% RSLogix 500 project DDE_Conecction_Excel.RSS, saved by version 8.30.00.16 %
PROJECT "UNTITLED"    % processor: Bul.1763 MicroLogix 1100 Series B %

PROGRAM FILES
  LAD 2 "MAIN"  4 rungs
  LAD 3 "DDE EXCEL"  31 rungs

DATA FILES
  O0 OUTPUT  4 elements
  I1 INPUT  6 elements
  S2 STATUS  66 elements
  B3 BINARY  2 elements
  T4 TIMER  8 elements
  C5 COUNTER  4 elements
  R6 CONTROL  1 elements
  N7 INTEGER  9 elements
  F8 FLOAT  1 elements
  ST9 STRINGS  9 elements

LADDER 2 "MAIN"
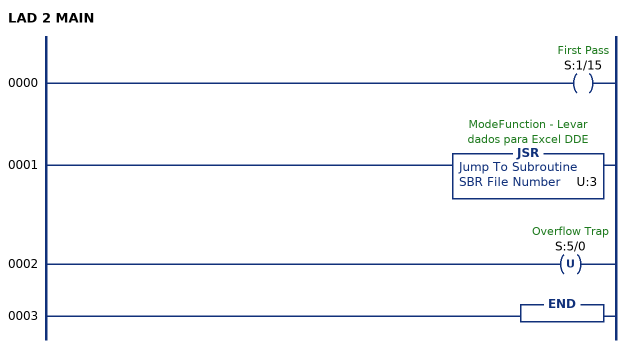
% Rung: 0 %
SOR OTE S:1/15 EOR
%   S:1/15  "First Pass" %
% Rung: 1 %
SOR JSR U:3 EOR
%   U:3  "ModeFunction - Levar dados para Excel DDE" %
% Rung: 2 %
SOR OTU S:5/0 EOR
%   S:5/0  "Overflow Trap" %
% Rung: 3 %
SOR END EOR

LADDER 3 "DDE EXCEL"
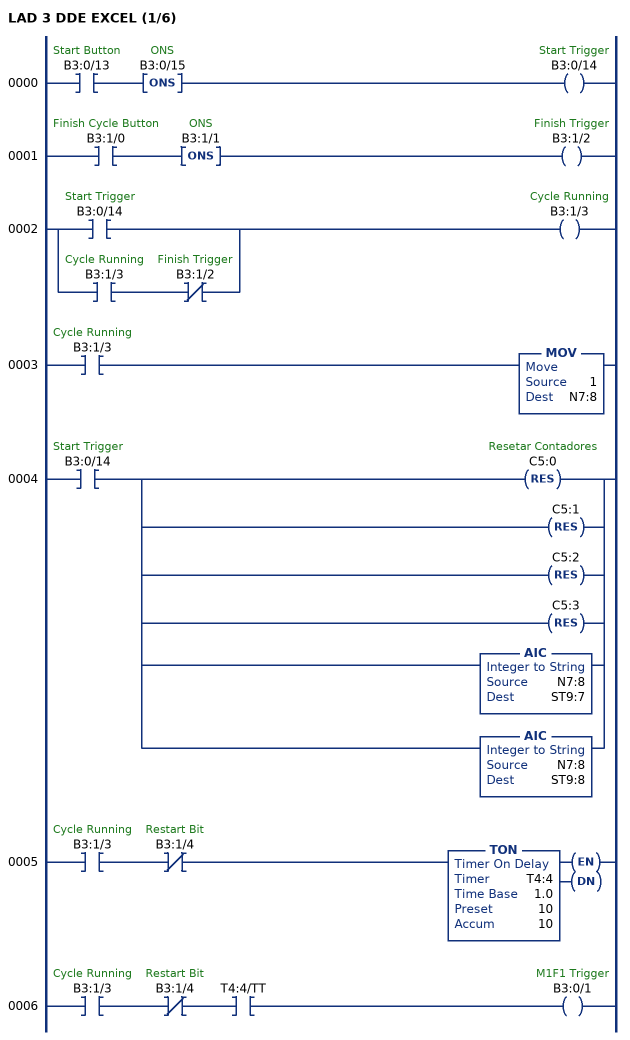
% Rung: 0 %
SOR XIC B3:0/13 ONS B3:0/15 OTE B3:0/14 EOR
%   B3:0/13  "Start Button" %
%   B3:0/15  "ONS" %
%   B3:0/14  "Start Trigger" %
% Rung: 1 %
SOR XIC B3:1/0 ONS B3:1/1 OTE B3:1/2 EOR
%   B3:1/0  "Finish Cycle Button" %
%   B3:1/1  "ONS" %
%   B3:1/2  "Finish Trigger" %
% Rung: 2 %
SOR BST XIC B3:0/14 NXB XIC B3:1/3 XIO B3:1/2 BND OTE B3:1/3 EOR
%   B3:0/14  "Start Trigger" %
%   B3:1/3  "Cycle Running" %
%   B3:1/2  "Finish Trigger" %
% Rung: 3 %
SOR XIC B3:1/3 MOV 1 N7:8 EOR
%   B3:1/3  "Cycle Running" %
% Rung: 4 %
SOR XIC B3:0/14 BST RES C5:0 NXB RES C5:1 NXB RES C5:2 NXB RES C5:3 NXB AIC N7:8 ST9:7 NXB AIC N7:8 ST9:8 BND EOR
%   B3:0/14  "Start Trigger" %
%   C5:0  "Resetar Contadores" %
% Rung: 5 %
SOR XIC B3:1/3 XIO B3:1/4 TON T4:4 1.0 10 10 EOR
%   B3:1/3  "Cycle Running" %
%   B3:1/4  "Restart Bit" %
% Rung: 6 %
SOR XIC B3:1/3 XIO B3:1/4 XIC T4:4/TT OTE B3:0/1 EOR
%   B3:1/3  "Cycle Running" %
%   B3:1/4  "Restart Bit" %
%   B3:0/1  "M1F1 Trigger" %

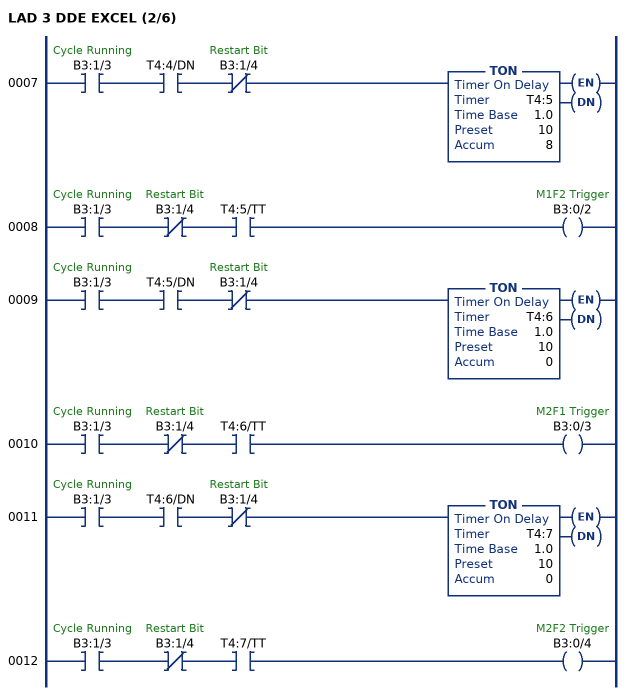
% Rung: 7 %
SOR XIC B3:1/3 XIC T4:4/DN XIO B3:1/4 TON T4:5 1.0 10 8 EOR
%   B3:1/3  "Cycle Running" %
%   B3:1/4  "Restart Bit" %
% Rung: 8 %
SOR XIC B3:1/3 XIO B3:1/4 XIC T4:5/TT OTE B3:0/2 EOR
%   B3:1/3  "Cycle Running" %
%   B3:1/4  "Restart Bit" %
%   B3:0/2  "M1F2 Trigger" %
% Rung: 9 %
SOR XIC B3:1/3 XIC T4:5/DN XIO B3:1/4 TON T4:6 1.0 10 0 EOR
%   B3:1/3  "Cycle Running" %
%   B3:1/4  "Restart Bit" %
% Rung: 10 %
SOR XIC B3:1/3 XIO B3:1/4 XIC T4:6/TT OTE B3:0/3 EOR
%   B3:1/3  "Cycle Running" %
%   B3:1/4  "Restart Bit" %
%   B3:0/3  "M2F1 Trigger" %
% Rung: 11 %
SOR XIC B3:1/3 XIC T4:6/DN XIO B3:1/4 TON T4:7 1.0 10 0 EOR
%   B3:1/3  "Cycle Running" %
%   B3:1/4  "Restart Bit" %
% Rung: 12 %
SOR XIC B3:1/3 XIO B3:1/4 XIC T4:7/TT OTE B3:0/4 EOR
%   B3:1/3  "Cycle Running" %
%   B3:1/4  "Restart Bit" %
%   B3:0/4  "M2F2 Trigger" %

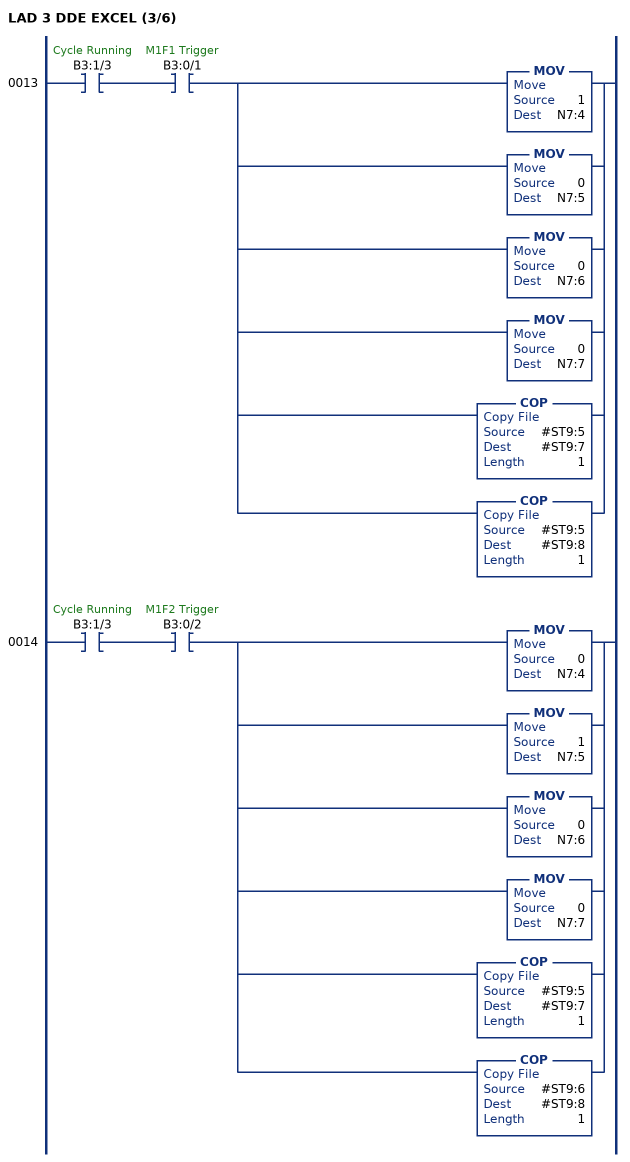
% Rung: 13 %
SOR XIC B3:1/3 XIC B3:0/1 BST MOV 1 N7:4 NXB MOV 0 N7:5 NXB MOV 0 N7:6 NXB MOV 0 N7:7 NXB COP #ST9:5 #ST9:7 1 NXB COP #ST9:5 #ST9:8 1 BND EOR
%   B3:1/3  "Cycle Running" %
%   B3:0/1  "M1F1 Trigger" %
% Rung: 14 %
SOR XIC B3:1/3 XIC B3:0/2 BST MOV 0 N7:4 NXB MOV 1 N7:5 NXB MOV 0 N7:6 NXB MOV 0 N7:7 NXB COP #ST9:5 #ST9:7 1 NXB COP #ST9:6 #ST9:8 1 BND EOR
%   B3:1/3  "Cycle Running" %
%   B3:0/2  "M1F2 Trigger" %

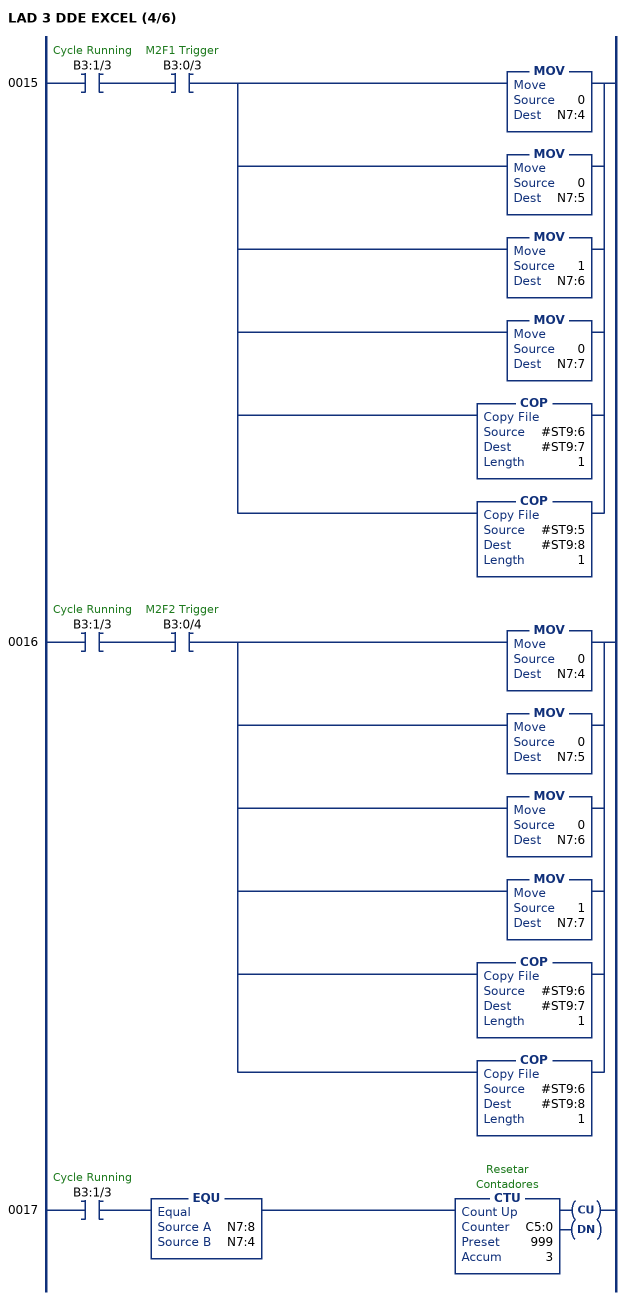
% Rung: 15 %
SOR XIC B3:1/3 XIC B3:0/3 BST MOV 0 N7:4 NXB MOV 0 N7:5 NXB MOV 1 N7:6 NXB MOV 0 N7:7 NXB COP #ST9:6 #ST9:7 1 NXB COP #ST9:5 #ST9:8 1 BND EOR
%   B3:1/3  "Cycle Running" %
%   B3:0/3  "M2F1 Trigger" %
% Rung: 16 %
SOR XIC B3:1/3 XIC B3:0/4 BST MOV 0 N7:4 NXB MOV 0 N7:5 NXB MOV 0 N7:6 NXB MOV 1 N7:7 NXB COP #ST9:6 #ST9:7 1 NXB COP #ST9:6 #ST9:8 1 BND EOR
%   B3:1/3  "Cycle Running" %
%   B3:0/4  "M2F2 Trigger" %
% Rung: 17 %
SOR XIC B3:1/3 EQU N7:8 N7:4 CTU C5:0 999 3 EOR
%   B3:1/3  "Cycle Running" %
%   C5:0  "Resetar Contadores" %

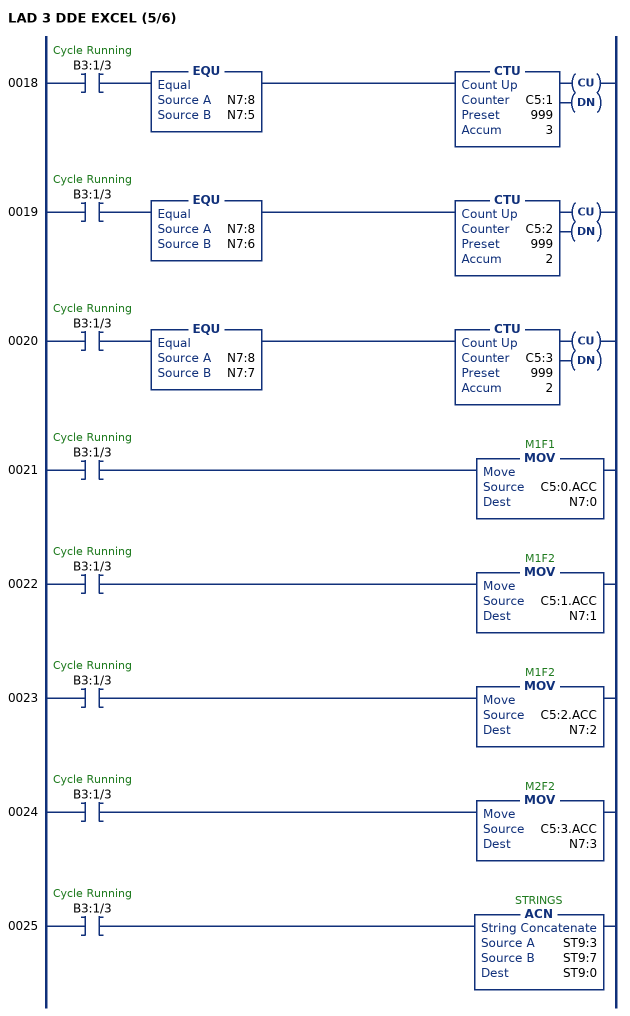
% Rung: 18 %
SOR XIC B3:1/3 EQU N7:8 N7:5 CTU C5:1 999 3 EOR
%   B3:1/3  "Cycle Running" %
% Rung: 19 %
SOR XIC B3:1/3 EQU N7:8 N7:6 CTU C5:2 999 2 EOR
%   B3:1/3  "Cycle Running" %
% Rung: 20 %
SOR XIC B3:1/3 EQU N7:8 N7:7 CTU C5:3 999 2 EOR
%   B3:1/3  "Cycle Running" %
% Rung: 21 %
SOR XIC B3:1/3 MOV C5:0.ACC N7:0 EOR
%   B3:1/3  "Cycle Running" %
%   C5:0  "Resetar Contadores" %
%   N7:0  "M1F1" %
% Rung: 22 %
SOR XIC B3:1/3 MOV C5:1.ACC N7:1 EOR
%   B3:1/3  "Cycle Running" %
%   N7:1  "M1F2" %
% Rung: 23 %
SOR XIC B3:1/3 MOV C5:2.ACC N7:2 EOR
%   B3:1/3  "Cycle Running" %
%   N7:2  "M1F2" %
% Rung: 24 %
SOR XIC B3:1/3 MOV C5:3.ACC N7:3 EOR
%   B3:1/3  "Cycle Running" %
%   N7:3  "M2F2" %
% Rung: 25 %
SOR XIC B3:1/3 ACN ST9:3 ST9:7 ST9:0 EOR
%   B3:1/3  "Cycle Running" %
%   ST9:0  STRINGS %

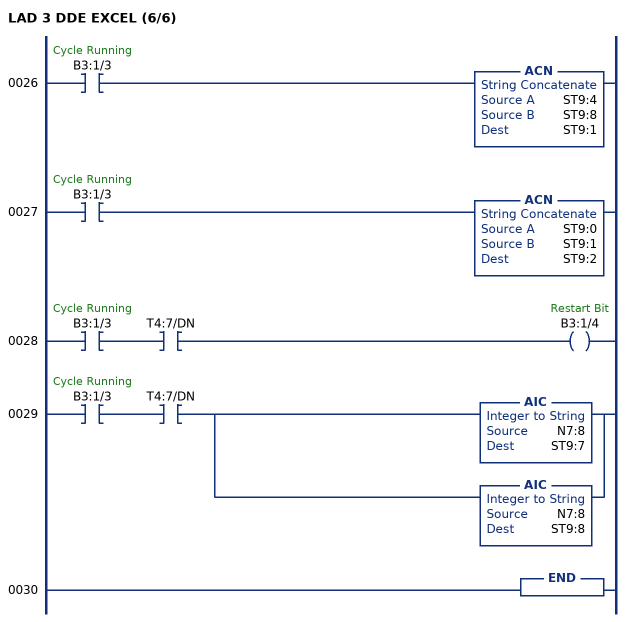
% Rung: 26 %
SOR XIC B3:1/3 ACN ST9:4 ST9:8 ST9:1 EOR
%   B3:1/3  "Cycle Running" %
% Rung: 27 %
SOR XIC B3:1/3 ACN ST9:0 ST9:1 ST9:2 EOR
%   B3:1/3  "Cycle Running" %
%   ST9:0  STRINGS %
% Rung: 28 %
SOR XIC B3:1/3 XIC T4:7/DN OTE B3:1/4 EOR
%   B3:1/3  "Cycle Running" %
%   B3:1/4  "Restart Bit" %
% Rung: 29 %
SOR XIC B3:1/3 XIC T4:7/DN BST AIC N7:8 ST9:7 NXB AIC N7:8 ST9:8 BND EOR
%   B3:1/3  "Cycle Running" %
% Rung: 30 %
SOR END EOR

OTHER DOCUMENTED ADDRESSES
  B3:0/5  "M1F1 Button"
  B3:0/6  "M1F2 Button"
  B3:0/7  "M2F1 Button"
  B3:0/8  "M2F2 Button"
  B3:0/9  "ONS"
  B3:0/10  "ONS"
  B3:0/11  "ONS"
  B3:0/12  "ONS"

DATA TABLE (non-zero values as saved)
DATA B3
% B3:0 % 0XA004 0X0008
DATA T4
% .PRE .ACC %
% T4:1 % 9999 0
% T4:2 % 9999 0
% T4:3 % 9999 0
% T4:4 % 10 10
% T4:5 % 10 8
% T4:6 % 10 0
% T4:7 % 10 0
DATA C5
% .PRE .ACC %
% C5:0 % 999 3
% C5:1 % 999 3
% C5:2 % 999 2
% C5:3 % 999 2
DATA N7
% N7:0 % 3 3 2 2 0 1 0 0 1
DATA ST9
% ST9:0 % "M1"
% ST9:1 % "F2"
% ST9:2 % "M1F2"
% ST9:3 % "M"
% ST9:4 % "F"
% ST9:5 % "1"
% ST9:6 % "2"
% ST9:7 % "1"
% ST9:8 % "2"
